// TIA Portal V19 export
DATA_BLOCK "Config"   // DB93
// stored: Access Published, MemoryReserve 100, Namespace Unit2.EM4
   VAR
      em { ExternalWritable := 'False'} : "LAF_typeEmConfiguration";   // Configuration of EM Parameters
      axis { ExternalWritable := 'False'} : Array[1.._.U2EM4_NO_OF_AXES] of DB_ANY;   // Assign the axis of the EM
      em4Parameters : "LAF_typeXyzhandlingEm4Parameters";
   END_VAR
BEGIN
   em.referenceDesignator.parent := WSTRING#'U1';
   em.referenceDesignator.relative := WSTRING#'EM1';
   // em4Parameters.cm1Axis119 : X
   // em4Parameters.cm1Axis119.production.distanceList[0] : 24 cells[0][0]constraintPosition
   // em4Parameters.cm1Axis119.production.distanceList[1] : 24 cells[0][-1]constraintPosition
   // em4Parameters.cm1Axis119.production.distanceList[2] : 24 cells[1][0]constraintPosition
   // em4Parameters.cm1Axis119.production.distanceList[3] : 36 cells[0][0]constraintPosition
   // em4Parameters.cm1Axis119.production.distanceList[4] : 36 cells[0][-1]constraintPosition
   // em4Parameters.cm1Axis119.production.distanceList[5] : 36 cells[1][0]constraintPosition
   // em4Parameters.cm1Axis119.production.distanceList[6] : Structure for a Position set point
   // em4Parameters.cm1Axis119.production.distanceList[7] : Structure for a Position set point
   // em4Parameters.cm1Axis119.production.distanceList[8] : Structure for a Position set point
   // em4Parameters.cm1Axis119.production.distanceList[9] : Structure for a Position set point
   // em4Parameters.cm1Axis119.production.distanceList[10] : 24 cells[0][0]plasticPosition
   // em4Parameters.cm1Axis119.production.distanceList[11] : 24 cells[0][-1]plasticPosition
   // em4Parameters.cm1Axis119.production.distanceList[12] : 24 cells[1][0]plasticPosition
   // em4Parameters.cm1Axis119.production.distanceList[13] : 36 cells[0][0]plasticPosition
   // em4Parameters.cm1Axis119.production.distanceList[14] : 36 cells[0][-1]plasticPosition
   // em4Parameters.cm1Axis119.production.distanceList[15] : 36 cells[1][0]plasticPosition
   // em4Parameters.cm1Axis119.production.distanceList[16] : Structure for a Position set point
   // em4Parameters.cm1Axis119.production.distanceList[17] : Structure for a Position set point
   // em4Parameters.cm1Axis119.production.distanceList[18] : Structure for a Position set point
   // em4Parameters.cm1Axis119.production.distanceList[19] : Structure for a Position set point
   // em4Parameters.cm1Axis119.production.distanceList[20] : ngConveyorPostion
   // em4Parameters.cm1Axis119.production.distanceList[21] : Structure for a Position set point
   // em4Parameters.cm1Axis119.production.distanceList[22] : Structure for a Position set point
   // em4Parameters.cm1Axis119.production.distanceList[23] : Structure for a Position set point
   // em4Parameters.cm1Axis119.production.distanceList[24] : Structure for a Position set point
   // em4Parameters.cm1Axis119.production.distanceList[25] : Structure for a Position set point
   // em4Parameters.cm1Axis119.production.distanceList[26] : Structure for a Position set point
   // em4Parameters.cm1Axis119.production.distanceList[27] : Structure for a Position set point
   // em4Parameters.cm1Axis119.production.distanceList[28] : Structure for a Position set point
   // em4Parameters.cm1Axis119.production.distanceList[29] : Structure for a Position set point
   // em4Parameters.cm1Axis119.production.distanceList[30] : 24电芯 拘束第一次抓取
   // em4Parameters.cm1Axis119.production.distanceList[31] : 24电芯 拘束第二次抓取
   // em4Parameters.cm1Axis119.production.distanceList[32] : 24电芯 拘束第三次抓取
   // em4Parameters.cm1Axis119.production.distanceList[33] : Structure for a Position set point
   // em4Parameters.cm1Axis119.production.distanceList[34] : Structure for a Position set point
   // em4Parameters.cm1Axis119.production.distanceList[35] : Structure for a Position set point
   // em4Parameters.cm1Axis119.production.distanceList[36] : Structure for a Position set point
   // em4Parameters.cm1Axis119.production.distanceList[37] : Structure for a Position set point
   // em4Parameters.cm1Axis119.production.distanceList[38] : Structure for a Position set point
   // em4Parameters.cm1Axis119.production.distanceList[39] : Structure for a Position set point
   // em4Parameters.cm1Axis119.production.distanceList[40] : 36电芯 拘束第1次抓取
   // em4Parameters.cm1Axis119.production.distanceList[41] : 36电芯 拘束第2次抓取
   // em4Parameters.cm1Axis119.production.distanceList[42] : 36电芯 拘束第3次抓取
   // em4Parameters.cm1Axis119.production.distanceList[43] : 36电芯 拘束第4次抓取
   // em4Parameters.cm1Axis119.production.distanceList[44] : 36电芯 拘束第5次抓取
   // em4Parameters.cm1Axis119.production.distanceList[45] : Structure for a Position set point
   // em4Parameters.cm1Axis119.production.distanceList[46] : Structure for a Position set point
   // em4Parameters.cm1Axis119.production.distanceList[47] : Structure for a Position set point
   // em4Parameters.cm1Axis119.production.distanceList[48] : Structure for a Position set point
   // em4Parameters.cm1Axis119.production.distanceList[49] : Structure for a Position set point
   // em4Parameters.cm1Axis119.production.distanceList[50] : 24电芯 塑料第一次抓放
   // em4Parameters.cm1Axis119.production.distanceList[51] : 24电芯 塑料第二次抓放
   // em4Parameters.cm1Axis119.production.distanceList[52] : 24电芯 塑料第三次抓放
   // em4Parameters.cm1Axis119.production.distanceList[53] : Structure for a Position set point
   // em4Parameters.cm1Axis119.production.distanceList[54] : Structure for a Position set point
   // em4Parameters.cm1Axis119.production.distanceList[55] : Structure for a Position set point
   // em4Parameters.cm1Axis119.production.distanceList[56] : Structure for a Position set point
   // em4Parameters.cm1Axis119.production.distanceList[57] : Structure for a Position set point
   // em4Parameters.cm1Axis119.production.distanceList[58] : Structure for a Position set point
   // em4Parameters.cm1Axis119.production.distanceList[59] : Structure for a Position set point
   // em4Parameters.cm1Axis119.production.distanceList[60] : 36电芯 塑料第1次抓放
   // em4Parameters.cm1Axis119.production.distanceList[61] : 36电芯 塑料第2次抓放
   // em4Parameters.cm1Axis119.production.distanceList[62] : 36电芯 塑料第3次抓放
   // em4Parameters.cm1Axis119.production.distanceList[63] : 36电芯 塑料第4次抓放
   // em4Parameters.cm1Axis119.production.distanceList[64] : 36电芯 塑料第5次抓放
   em4Parameters.cm1Axis119.production.distanceList[0].position := 30.0;
   em4Parameters.cm1Axis119.production.distanceList[1].position := 150.0;
   em4Parameters.cm1Axis119.production.distanceList[2..3].position := 30.0;
   em4Parameters.cm1Axis119.production.distanceList[4].position := 190.0;
   em4Parameters.cm1Axis119.production.distanceList[5].position := 30.0;
   em4Parameters.cm1Axis119.production.distanceList[10].position := 45.0;
   em4Parameters.cm1Axis119.production.distanceList[11].position := 165.0;
   em4Parameters.cm1Axis119.production.distanceList[12..13].position := 45.0;
   em4Parameters.cm1Axis119.production.distanceList[14].position := 225.0;
   em4Parameters.cm1Axis119.production.distanceList[15].position := 45.0;
   em4Parameters.cm1Axis119.production.distanceList[20].position := 45.0;
   em4Parameters.cm1Axis119.production.distanceList[0..5].velocity := 30.0;
   em4Parameters.cm1Axis119.production.distanceList[10..15].velocity := 30.0;
   em4Parameters.cm1Axis119.production.distanceList[20].velocity := 30.0;
   // em4Parameters.cm2Axis120 : Y
   // em4Parameters.cm2Axis120.production.distanceList[0] : 24 cells[0][0]constraintPosition
   // em4Parameters.cm2Axis120.production.distanceList[1] : 24 cells[0][-1]constraintPosition
   // em4Parameters.cm2Axis120.production.distanceList[2] : 24 cells[1][0]constraintPosition
   // em4Parameters.cm2Axis120.production.distanceList[3] : 36 cells[0][0]constraintPosition
   // em4Parameters.cm2Axis120.production.distanceList[4] : 36 cells[0][-1]constraintPosition
   // em4Parameters.cm2Axis120.production.distanceList[5] : 36 cells[1][0]constraintPosition
   // em4Parameters.cm2Axis120.production.distanceList[6] : Structure for a Position set point
   // em4Parameters.cm2Axis120.production.distanceList[7] : Structure for a Position set point
   // em4Parameters.cm2Axis120.production.distanceList[8] : Structure for a Position set point
   // em4Parameters.cm2Axis120.production.distanceList[9] : Structure for a Position set point
   // em4Parameters.cm2Axis120.production.distanceList[10] : 24 cells[0][0]plasticPosition
   // em4Parameters.cm2Axis120.production.distanceList[11] : 24 cells[0][-1]plasticPosition
   // em4Parameters.cm2Axis120.production.distanceList[12] : 24 cells[1][0]plasticPosition
   // em4Parameters.cm2Axis120.production.distanceList[13] : 36 cells[0][0]plasticPosition
   // em4Parameters.cm2Axis120.production.distanceList[14] : 36 cells[0][-1]plasticPosition
   // em4Parameters.cm2Axis120.production.distanceList[15] : 36 cells[1][0]plasticPosition
   // em4Parameters.cm2Axis120.production.distanceList[16] : Structure for a Position set point
   // em4Parameters.cm2Axis120.production.distanceList[17] : Structure for a Position set point
   // em4Parameters.cm2Axis120.production.distanceList[18] : Structure for a Position set point
   // em4Parameters.cm2Axis120.production.distanceList[19] : Structure for a Position set point
   // em4Parameters.cm2Axis120.production.distanceList[20] : ngConveyorPostion
   em4Parameters.cm2Axis120.production.distanceList[0..1].position := 40.0;
   em4Parameters.cm2Axis120.production.distanceList[2].position := 60.0;
   em4Parameters.cm2Axis120.production.distanceList[3..4].position := 50.0;
   em4Parameters.cm2Axis120.production.distanceList[5].position := 70.0;
   em4Parameters.cm2Axis120.production.distanceList[10..11].position := 180.0;
   em4Parameters.cm2Axis120.production.distanceList[12].position := 200.0;
   em4Parameters.cm2Axis120.production.distanceList[13..14].position := 190.0;
   em4Parameters.cm2Axis120.production.distanceList[15].position := 210.0;
   em4Parameters.cm2Axis120.production.distanceList[20].position := 300.0;
   em4Parameters.cm2Axis120.production.distanceList[0..5].velocity := 30.0;
   em4Parameters.cm2Axis120.production.distanceList[10..15].velocity := 30.0;
   em4Parameters.cm2Axis120.production.distanceList[20].velocity := 30.0;
   // em4Parameters.cm3Axis121 : Z
   // em4Parameters.cm3Axis121.production.distanceList[0] : 24 cells[0][0]constraintPosition
   // em4Parameters.cm3Axis121.production.distanceList[1] : 24 cells[0][-1]constraintPosition
   // em4Parameters.cm3Axis121.production.distanceList[2] : 24 cells[1][0]constraintPosition
   // em4Parameters.cm3Axis121.production.distanceList[3] : 36 cells[0][0]constraintPosition
   // em4Parameters.cm3Axis121.production.distanceList[4] : 36 cells[0][-1]constraintPosition
   // em4Parameters.cm3Axis121.production.distanceList[5] : 36 cells[1][0]constraintPosition
   // em4Parameters.cm3Axis121.production.distanceList[6] : Structure for a Position set point
   // em4Parameters.cm3Axis121.production.distanceList[7] : Structure for a Position set point
   // em4Parameters.cm3Axis121.production.distanceList[8] : Structure for a Position set point
   // em4Parameters.cm3Axis121.production.distanceList[9] : Structure for a Position set point
   // em4Parameters.cm3Axis121.production.distanceList[10] : 24 cells[0][0]plasticPosition
   // em4Parameters.cm3Axis121.production.distanceList[11] : 24 cells[0][-1]plasticPosition
   // em4Parameters.cm3Axis121.production.distanceList[12] : 24 cells[1][0]plasticPosition
   // em4Parameters.cm3Axis121.production.distanceList[13] : 36 cells[0][0]plasticPosition
   // em4Parameters.cm3Axis121.production.distanceList[14] : 36 cells[0][-1]plasticPosition
   // em4Parameters.cm3Axis121.production.distanceList[15] : 36 cells[1][0]plasticPosition
   // em4Parameters.cm3Axis121.production.distanceList[16] : Structure for a Position set point
   // em4Parameters.cm3Axis121.production.distanceList[17] : Structure for a Position set point
   // em4Parameters.cm3Axis121.production.distanceList[18] : Structure for a Position set point
   // em4Parameters.cm3Axis121.production.distanceList[19] : Structure for a Position set point
   // em4Parameters.cm3Axis121.production.distanceList[20] : ngConveyorPostion
   em4Parameters.cm3Axis121.production.distanceList[0..5].position := 90.0;
   em4Parameters.cm3Axis121.production.distanceList[10..15].position := 90.0;
   em4Parameters.cm3Axis121.production.distanceList[20].position := 100.0;
   em4Parameters.cm3Axis121.production.distanceList[0..5].velocity := 30.0;
   em4Parameters.cm3Axis121.production.distanceList[10..15].velocity := 30.0;
   em4Parameters.cm3Axis121.production.distanceList[20].velocity := 30.0;
END_DATA_BLOCK
